(* Logix 5000 project; controller ACMI_PLC vendor 1 type 14 code 101 rev 19.11; software revision 19.01; part 8 of 9 *)
(* tags used below, declared in another part *)
   A : DINT;
   ACMI_BR_CNT : DINT;
   ACMI_Stat_Size : INT;
   ACMI_TO_CNT : DINT;
   ADCA : DINT;
   ADCB : DINT;
   B : DINT;
   Beam_MaxQ : DINT;
   Beam_MinQ : DINT;
   Beam_Q : DINT;
   BR_Stack : DINT[7200];
   BR_Stack_MAX : DINT;
   BR_Stack_Sum : DINT;
   BR_Stack_Top : DINT;
   BSSS_CLOSED : ALIAS FOR PointIONet:7:I.Pt00Data;
   BYPASS_KEY : ALIAS FOR PointIONet:5:I.Pt07Data;
   FAULT_BEAM_BL : BOOL;
   FAULT_BEAM_HI : BOOL;
   FAULT_BEAM_LO : BOOL;
   FAULT_BR_ACC : BOOL;
   FAULT_CODE : DINT;
   FAULT_QOW1 : BOOL;
   FAULT_ST1_AB_HI : BOOL;
   FAULT_ST1_AB_LO : BOOL;
   FAULT_ST1_BA_HI : BOOL;
   FAULT_ST1_BA_LO : BOOL;
   FAULT_ST1_BLA : BOOL;
   FAULT_ST1_BLB : BOOL;
   FAULT_ST1_QAT : BOOL;
   FAULT_ST2_AB_HI : BOOL;
   FAULT_ST2_AB_LO : BOOL;
   FAULT_ST2_BA_HI : BOOL;
   FAULT_ST2_BA_LO : BOOL;
   FAULT_ST2_BLA : BOOL;
   FAULT_ST2_BLB : BOOL;
   FAULT_ST2_QAT : BOOL;
   FAULT_TO_ACC : BOOL;
   FAULT_TWB : BOOL;
   FAULT_WDT : BOOL;
   Initialize : BOOL;
   LBSS_CLOSED : ALIAS FOR PointIONet:7:I.Pt01Data;
   ST1_MaxQ : DINT;
   ST1_MinQ : DINT;
   ST1_QAB : DINT;
   ST1_QBA : DINT;
   ST2_MaxQ : DINT;
   ST2_MinQ : DINT;
   ST2_QAB : DINT;
   ST2_QBA : DINT;
   ST_HI_FAULT : BOOL;
   ST_LO_FAULT : BOOL;
   ST_Size : BOOL;
   ST_Type : BOOL;
   Stack_Size : DINT;
   TO_Cntr : COUNTER;
   TO_DISABLED : ALIAS FOR PointIONet:7:I.Pt03Data;
   TO_Stack : DINT[120];
   TO_Stack_MAX : DINT;
   TO_Stack_Size : DINT;
   TO_Stack_Sum : DINT;
   TO_Stack_Top : DINT;
   TO_Status_Error : BOOL;
   Update_ST1_QAB : BOOL;
   Update_ST1_QBA : BOOL;
   Update_ST2_QAB : BOOL;
   Update_ST2_QBA : BOOL;
   Zero : DINT[7200];

        [22].Hist[2930] := 1, [22].Hist[2938] := 1, [22].Hist[2946] := 1, [22].Hist[2954] := 1, [22].Hist[2962] := 1, [22].Hist[2970] := 1, [22].Hist[2975] := 1, [22].Hist[2978] := 1, [22].Hist[2986] := 1, [22].Hist[2994] := 1, [22].Hist[3002] := 1, [22].Hist[3010] := 1, [22].Hist[3018] := 1, [22].Hist[3026] := 1, [22].Hist[3034] := 1, [22].Hist[3042] := 1, [22].Hist[3050] := 1, [22].Hist[3058] := 1, [22].Hist[3066] := 1, [22].Hist[3074] := 1, [22].Hist[3082] := 1, [22].Hist[3090] := 1, [22].Hist[3098] := 1, [22].Hist[3106] := 1, [22].Hist[3114] := 1, [22].Hist[3122] := 1, [22].Hist[3130] := 1, [22].Hist[3138] := 1, [22].Hist[3146] := 1, [22].Hist[3152] := 1, [22].Hist[3154] := 1, [22].Hist[3162] := 1, [22].Hist[3170] := 1, [22].Hist[3178] := 1, [22].Hist[3181] := 1, [22].Hist[3186] := 1, [22].Hist[3194] := 1, [22].Hist[3202] := 1, [22].Hist[3210] := 1, [22].Hist[3218] := 1, [22].Hist[3226] := 1, [22].Hist[3234] := 1, [22].Hist[3242] := 1, [22].Hist[3250] := 1, [22].Hist[3258] := 1, [22].Hist[3266] := 1, [22].Hist[3274] := 1, [22].Hist[3282] := 1, [22].Hist[3290] := 1, [22].Hist[3298] := 1, [22].Hist[3306] := 1, [22].Hist[3314] := 1, [22].Hist[3322] := 1, [22].Hist[3330] := 1, [22].Hist[3333] := 1, [22].Hist[3338] := 1, [22].Hist[3346] := 1, [22].Hist[3354] := 1, [22].Hist[3362] := 1, [22].Hist[3370] := 1,
        [22].Hist[3378] := 1, [22].Hist[3386] := 1, [22].Hist[3394] := 1, [22].Hist[3402] := 1, [22].Hist[3410] := 1, [22].Hist[3418] := 1, [22].Hist[3420] := 1, [22].Hist[3426] := 1, [22].Hist[3434] := 1, [22].Hist[3442] := 1, [22].Hist[3450] := 1, [22].Hist[3458] := 1, [22].Hist[3466] := 1, [22].Hist[3474] := 1, [22].Hist[3482] := 1, [22].Hist[3490] := 1, [22].Hist[3497] := 1, [22].Hist[3498] := 1, [22].Hist[3506] := 1, [22].Hist[3514] := 1, [22].Hist[3522] := 1, [22].Hist[3530] := 1, [22].Hist[3538] := 1, [22].Hist[3546] := 1, [22].Hist[3554] := 1, [22].Hist[3562] := 1, [22].Hist[3570] := 1, [22].Hist[3578] := 1, [22].Hist[3586] := 1, [22].Hist[3594] := 1, [22].Hist[3602] := 1, [22].Hist[3610] := 1, [22].Hist[3618] := 1, [22].Hist[3626] := 1, [22].Hist[3634] := 1, [22].Hist[3642] := 1, [22].Hist[3650] := 1, [22].Hist[3658] := 1, [22].Hist[3666] := 1, [22].Hist[3674] := 1, [22].Hist[3682] := 1, [22].Hist[3690] := 1, [22].Hist[3698] := 1, [22].Hist[3706] := 1, [22].Hist[3714] := 1, [22].Hist[3722] := 1, [22].Hist[3730] := 1, [22].Hist[3738] := 1, [22].Hist[3746] := 1, [22].Hist[3754] := 1, [22].Hist[3762] := 1, [22].Hist[3770] := 1, [22].Hist[3778] := 1, [22].Hist[3786] := 1, [22].Hist[3794] := 1, [22].Hist[3802] := 1, [22].Hist[3810] := 1, [22].Hist[3818] := 1, [22].Hist[3826] := 1, [22].Hist[3834] := 1,
        [22].Hist[3842] := 1, [22].Hist[3850] := 1, [22].Hist[3858] := 1, [22].Hist[3866] := 1, [22].Hist[3874] := 1, [22].Hist[3882] := 1, [22].Hist[3890] := 1, [22].Hist[3898] := 1, [22].Hist[3906] := 1, [22].Hist[3914] := 1, [22].Hist[3922] := 1, [22].Hist[3924] := 1, [22].Hist[3930] := 1, [22].Hist[3938] := 1, [22].Hist[3946] := 1, [22].Hist[3954] := 1, [22].Hist[3962] := 1, [22].Hist[3970] := 1, [22].Hist[3978] := 1, [22].Hist[3986] := 1, [22].Hist[3994] := 1, [22].Hist[4002] := 1, [22].Hist[4010] := 1, [22].Hist[4018] := 1, [22].Hist[4026] := 1, [22].Hist[4034] := 1, [22].Hist[4042] := 1, [22].Hist[4045] := 1, [22].Hist[4050] := 1, [22].Hist[4058] := 1, [22].Hist[4066] := 1, [22].Hist[4074] := 1, [22].Hist[4082] := 1, [22].Hist[4090] := 1, [22].Top := 3955, [22].Sum := 539, [23].Hist[68] := 1, [23].Hist[123] := 1, [23].Hist[181] := 1, [23].Hist[417] := 1, [23].Hist[431] := 1, [23].Hist[488] := 1, [23].Hist[540] := 1, [23].Hist[567] := 1, [23].Hist[661] := 1, [23].Hist[805] := 1, [23].Hist[1153] := 1, [23].Hist[1377] := 1, [23].Hist[1435] := 1, [23].Hist[1727] := 1, [23].Hist[1773] := 1, [23].Hist[1817] := 1, [23].Hist[2324] := 1, [23].Hist[2512] := 1, [23].Hist[2756] := 1, [23].Hist[2975] := 1, [23].Hist[3152] := 1, [23].Hist[3181] := 1, [23].Hist[3333] := 1, [23].Hist[3420] := 1,
        [23].Hist[3497] := 1, [23].Hist[3924] := 1, [23].Hist[4045] := 1, [23].Top := 3955, [23].Sum := 27);
   Bx : DINT; {access Read Only}
   Data_Type : BOOL := 1;
   DrdyTimer : TIMER := (PRE := 500, ACC := 200, EN := 1, TT := 1);
   DrdyWDT : DINT := 220;
   ev_num : COUNTER := (ACC := 866343322, DN := 1);
   Fit_Linear_1 : DINT := 91449; {constant}
   Fit_Linear_2 : DINT := 10000; {constant}
   Fit_Off : DINT := 7; {constant}
   Fit_Quad_1 : DINT := 219; {constant}
   Fit_Quad_2 : DINT := 1000000; {constant}
   Hist : BOOL[4096] := ([956] := 1, [1408] := 1, [2824] := 1, [3245] := 1, [3333] := 1, [3825] := 1, [4017] := 1);
   index : DINT;
   NewData : BOOL := 1;
   Q : DINT := 15921;
   QIW : BOOL := 1;
   Qlinear : DINT := 15299;
   QOW_FailSafe : TIMER := (PRE := 2000, ACC := 340); {access Read Only}
   QOW_Latch : BOOL;
   Qquad : DINT := 615;
   ReadData : BOOL;
   Relay_Status : ALIAS FOR PointIONet:5:I.Pt04Data;
   Safety_Shutters : BOOL;
   ST1AB_ADCA : DINT := 64; {access Read Only}
   ST1AB_ADCB : DINT := 3; {access Read Only}
   ST1BA_ADCA : DINT := -1; {access Read Only}
   ST1BA_ADCB : DINT := 62; {access Read Only}
   ST2AB_ADCA : DINT := 1692; {access Read Only}
   ST2AB_ADCB : DINT := 3; {access Read Only}
   ST2BA_ADCA : DINT; {access Read Only}
   ST2BA_ADCB : DINT := 1673; {access Read Only}
   Stack_Data : DINT := 180;
   STQ : DINT := 15921; {access Read Only}
   STQmax : DINT := 16400; {access Read Only}
   STQmin : DINT := 15400; {access Read Only}
   Sum : INT := 7;
   Toggle : BitStat[12];
   Top : INT := 361;
   TWB_FailSafe : TIMER := (PRE := 2000, ACC := 20); {access Read Only}
   TWB_Latch : BOOL;
   Update_Latch : BOOL := 1; {access Read Only}
   Update_Unlatch : BOOL; {access Read Only}
   w1 : DINT; {access Read Only}
   w2 : DINT; {access Read Only}
   WDT_Event_Limit : DINT := 265; {constant, access Read Only}
   x : DINT := 1673;
   y : DINT;
   z : DINT := 1673;
   z2 : DINT;
END_VAR

ROUTINE Bit_Toggle   (* ladder *)
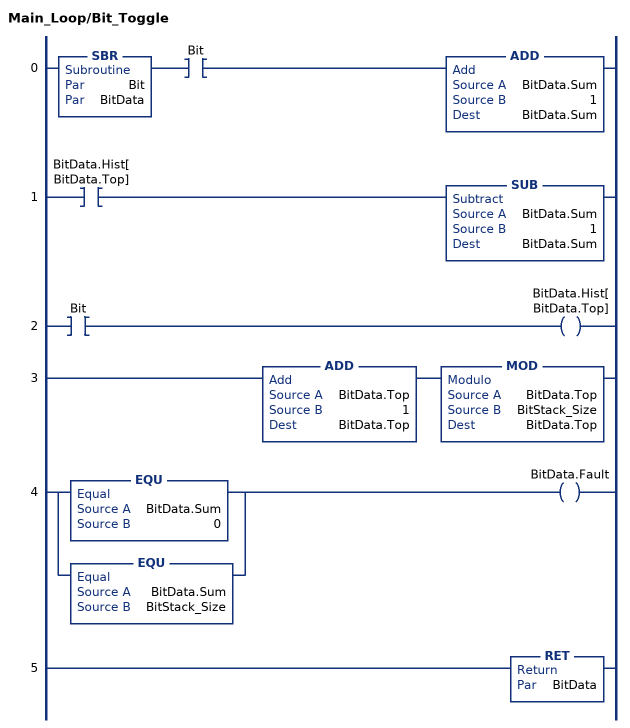
   [picture p14: Main_Loop/Bit_Toggle rungs 0-5]
   0: SBR(Bit,BitData)XIC(Bit)ADD(BitData.Sum,1,BitData.Sum);
   1: XIC(BitData.Hist[BitData.Top])SUB(BitData.Sum,1,BitData.Sum);
   2: XIC(Bit)OTE(BitData.Hist[BitData.Top]);
   3: ADD(BitData.Top,1,BitData.Top)MOD(BitData.Top,BitStack_Size,BitData.Top);
   4: [EQU(BitData.Sum,0) ,EQU(BitData.Sum,BitStack_Size) ]OTE(BitData.Fault);
   5: RET(BitData);
END_ROUTINE

ROUTINE Calc_Q   (* ladder *)
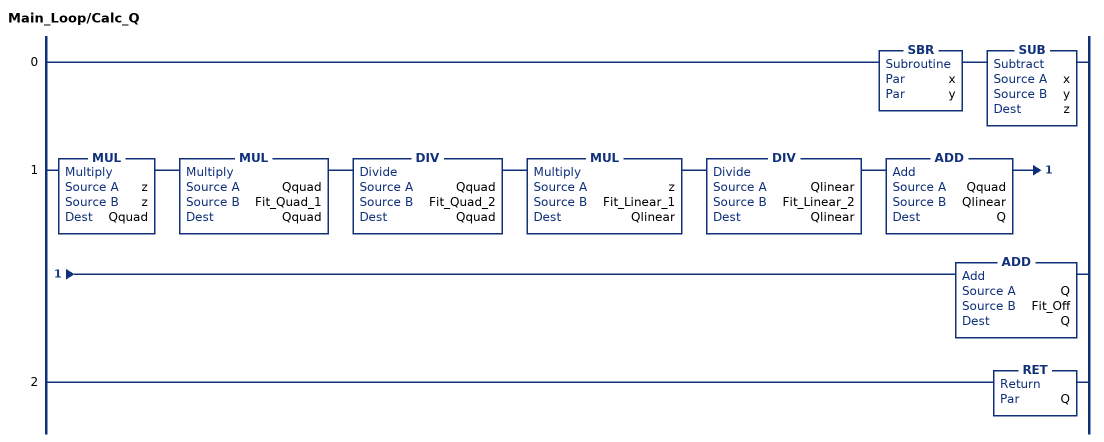
   0: SBR(x,y)SUB(x,y,z);
   1: MUL(z,z,Qquad)MUL(Qquad,Fit_Quad_1,Qquad)DIV(Qquad,Fit_Quad_2,Qquad)MUL(z,Fit_Linear_1,Qlinear)DIV(Qlinear,Fit_Linear_2,Qlinear)ADD(Qquad,Qlinear,Q)ADD(Q,Fit_Off,Q);
   2: RET(Q);
END_ROUTINE

ROUTINE MainRoutine   (* ladder *)
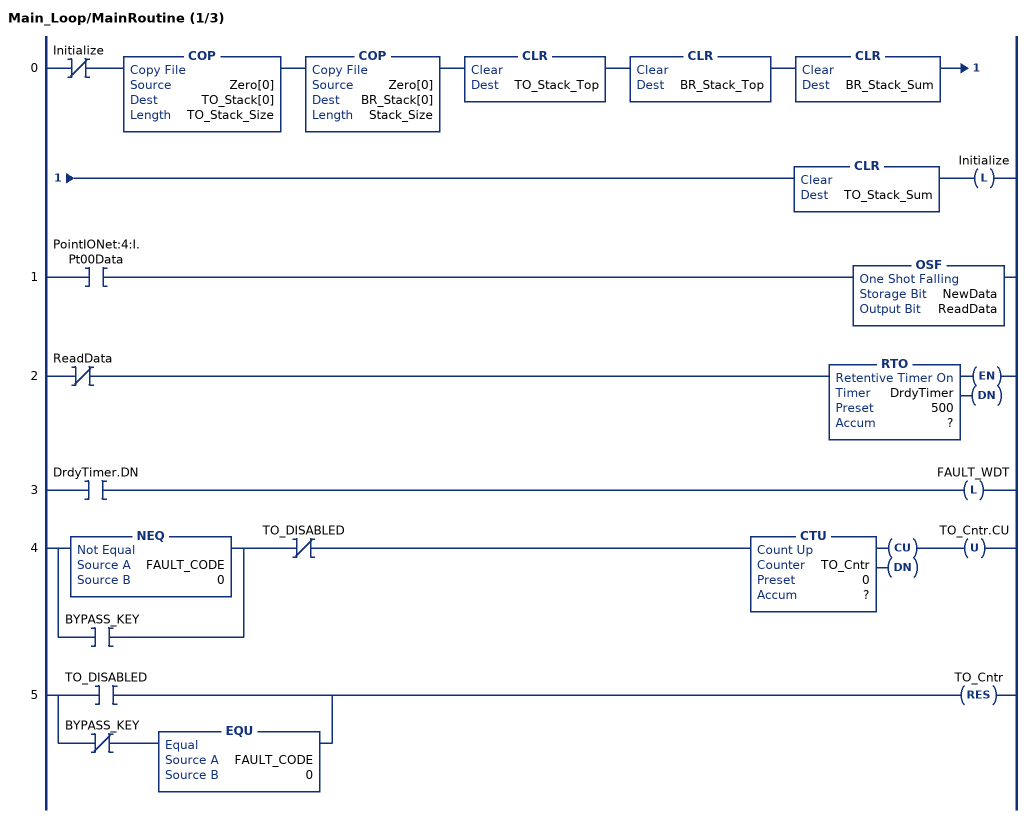
   0: XIO(Initialize)COP(Zero[0],TO_Stack[0],TO_Stack_Size)COP(Zero[0],BR_Stack[0],Stack_Size)CLR(TO_Stack_Top)CLR(BR_Stack_Top)CLR(BR_Stack_Sum)CLR(TO_Stack_Sum)OTL(Initialize);
   1: XIC(PointIONet:4:I.Pt00Data)OSF(NewData,ReadData);
   2: XIO(ReadData)RTO(DrdyTimer,?,?);
   3: XIC(DrdyTimer.DN)OTL(FAULT_WDT);
   4: [NEQ(FAULT_CODE,0) ,XIC(BYPASS_KEY) ]XIO(TO_DISABLED)CTU(TO_Cntr,?,?)OTU(TO_Cntr.CU);
   5: [XIC(TO_DISABLED) ,XIO(BYPASS_KEY) EQU(FAULT_CODE,0) ]RES(TO_Cntr);
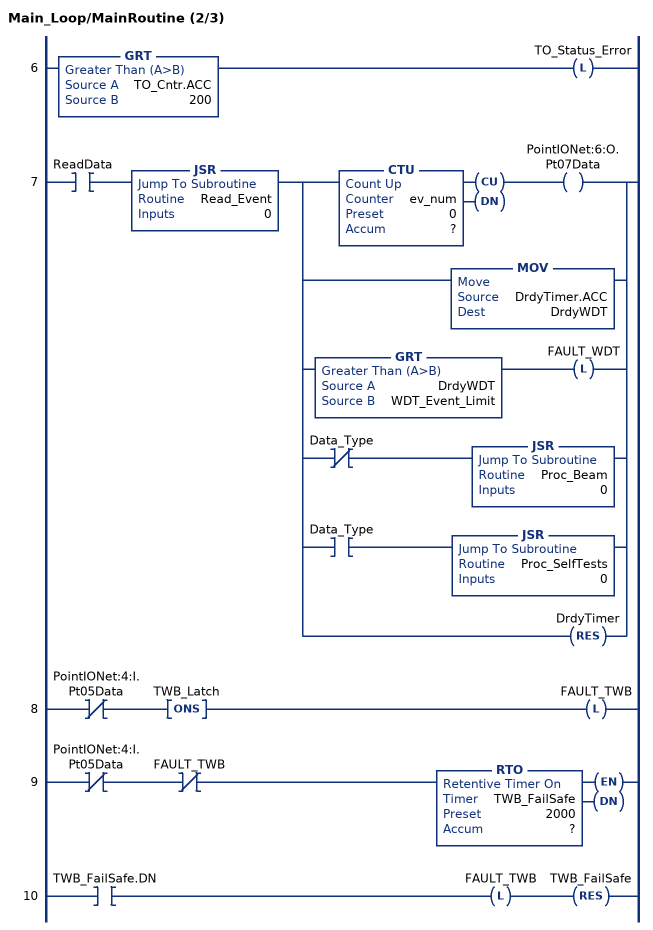
   6: GRT(TO_Cntr.ACC,200)OTL(TO_Status_Error);
   7: XIC(ReadData)JSR(Read_Event,0)[CTU(ev_num,?,?) OTE(PointIONet:6:O.Pt07Data) ,MOV(DrdyTimer.ACC,DrdyWDT) ,GRT(DrdyWDT,WDT_Event_Limit) OTL(FAULT_WDT) ,XIO(Data_Type) JSR(Proc_Beam,0) ,XIC(Data_Type) JSR(Proc_SelfTests,0) ,RES(DrdyTimer) ];
   8: XIO(PointIONet:4:I.Pt05Data)ONS(TWB_Latch)OTL(FAULT_TWB);
   9: XIO(PointIONet:4:I.Pt05Data)XIO(FAULT_TWB)RTO(TWB_FailSafe,?,?);
   10: XIC(TWB_FailSafe.DN)OTL(FAULT_TWB)RES(TWB_FailSafe);
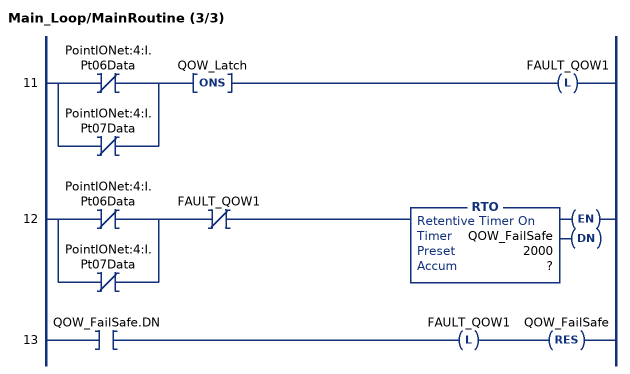
   11: [XIO(PointIONet:4:I.Pt06Data) ,XIO(PointIONet:4:I.Pt07Data) ]ONS(QOW_Latch)OTL(FAULT_QOW1);
   12: [XIO(PointIONet:4:I.Pt06Data) ,XIO(PointIONet:4:I.Pt07Data) ]XIO(FAULT_QOW1)RTO(QOW_FailSafe,?,?);
   13: XIC(QOW_FailSafe.DN)OTL(FAULT_QOW1)RES(QOW_FailSafe);
END_ROUTINE

ROUTINE Proc_Beam   (* ladder *)
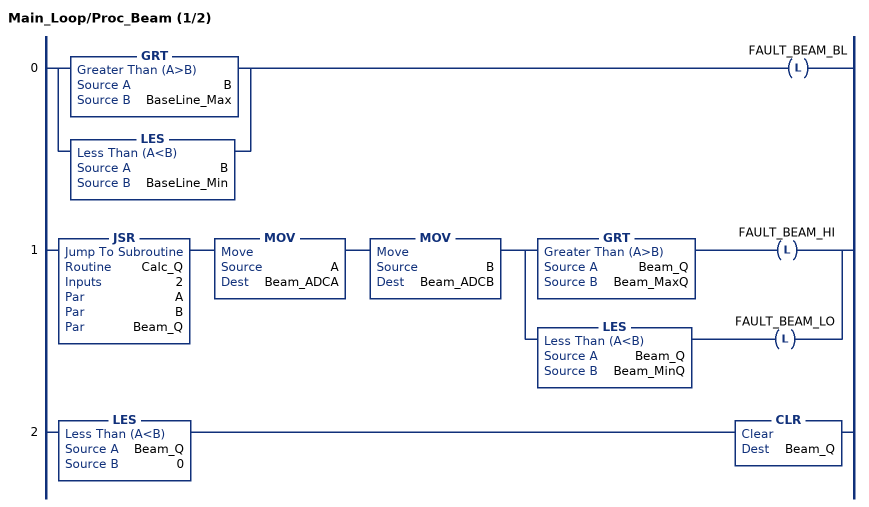
   0: [GRT(B,BaseLine_Max) ,LES(B,BaseLine_Min) ]OTL(FAULT_BEAM_BL);
   1: JSR(Calc_Q,2,A,B,Beam_Q)MOV(A,Beam_ADCA)MOV(B,Beam_ADCB)[GRT(Beam_Q,Beam_MaxQ) OTL(FAULT_BEAM_HI) ,LES(Beam_Q,Beam_MinQ) OTL(FAULT_BEAM_LO) ];
   2: LES(Beam_Q,0)CLR(Beam_Q);
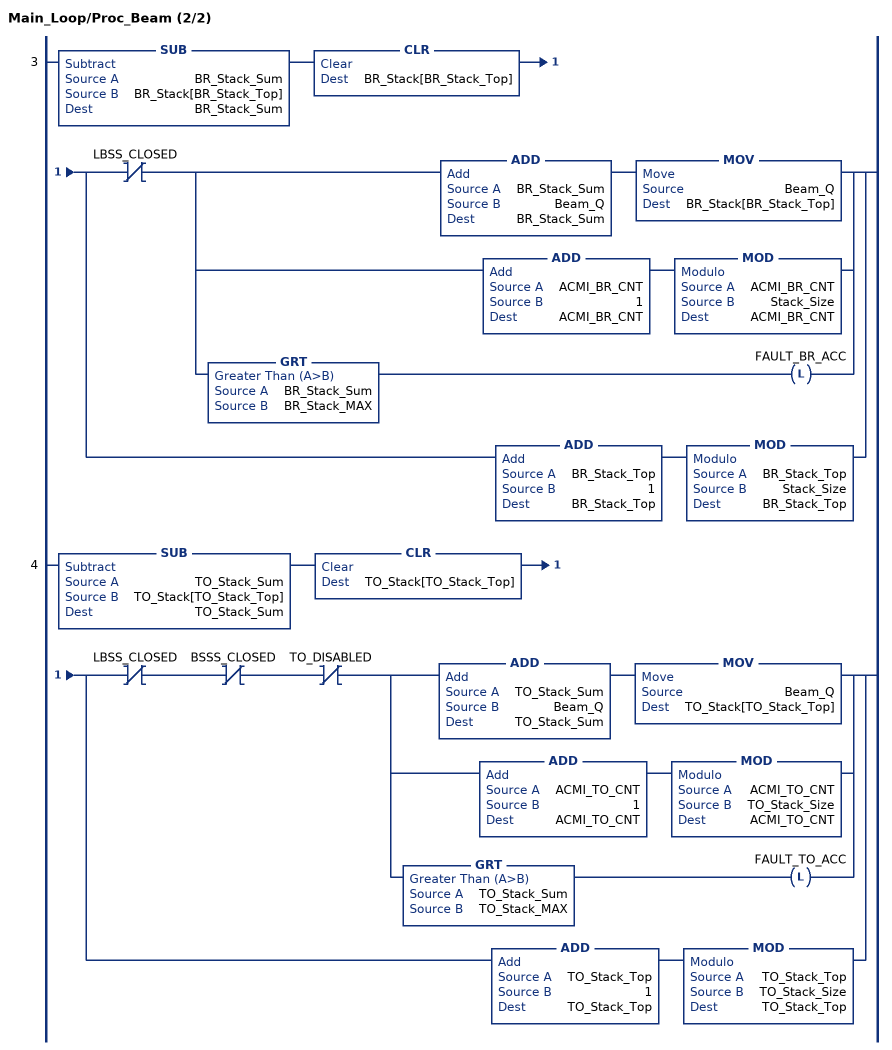
   3: SUB(BR_Stack_Sum,BR_Stack[BR_Stack_Top],BR_Stack_Sum)CLR(BR_Stack[BR_Stack_Top])[XIO(LBSS_CLOSED) [ADD(BR_Stack_Sum,Beam_Q,BR_Stack_Sum) MOV(Beam_Q,BR_Stack[BR_Stack_Top]) ,ADD(ACMI_BR_CNT,1,ACMI_BR_CNT) MOD(ACMI_BR_CNT,Stack_Size,ACMI_BR_CNT) ,GRT(BR_Stack_Sum,BR_Stack_MAX) OTL(FAULT_BR_ACC) ] ,ADD(BR_Stack_Top,1,BR_Stack_Top) MOD(BR_Stack_Top,Stack_Size,BR_Stack_Top) ];
   4: SUB(TO_Stack_Sum,TO_Stack[TO_Stack_Top],TO_Stack_Sum)CLR(TO_Stack[TO_Stack_Top])[XIO(LBSS_CLOSED) XIO(BSSS_CLOSED) XIO(TO_DISABLED) [ADD(TO_Stack_Sum,Beam_Q,TO_Stack_Sum) MOV(Beam_Q,TO_Stack[TO_Stack_Top]) ,ADD(ACMI_TO_CNT,1,ACMI_TO_CNT) MOD(ACMI_TO_CNT,TO_Stack_Size,ACMI_TO_CNT) ,GRT(TO_Stack_Sum,TO_Stack_MAX) OTL(FAULT_TO_ACC) ] ,ADD(TO_Stack_Top,1,TO_Stack_Top) MOD(TO_Stack_Top,TO_Stack_Size,TO_Stack_Top) ];
END_ROUTINE

ROUTINE Proc_SelfTests   (* ladder *)
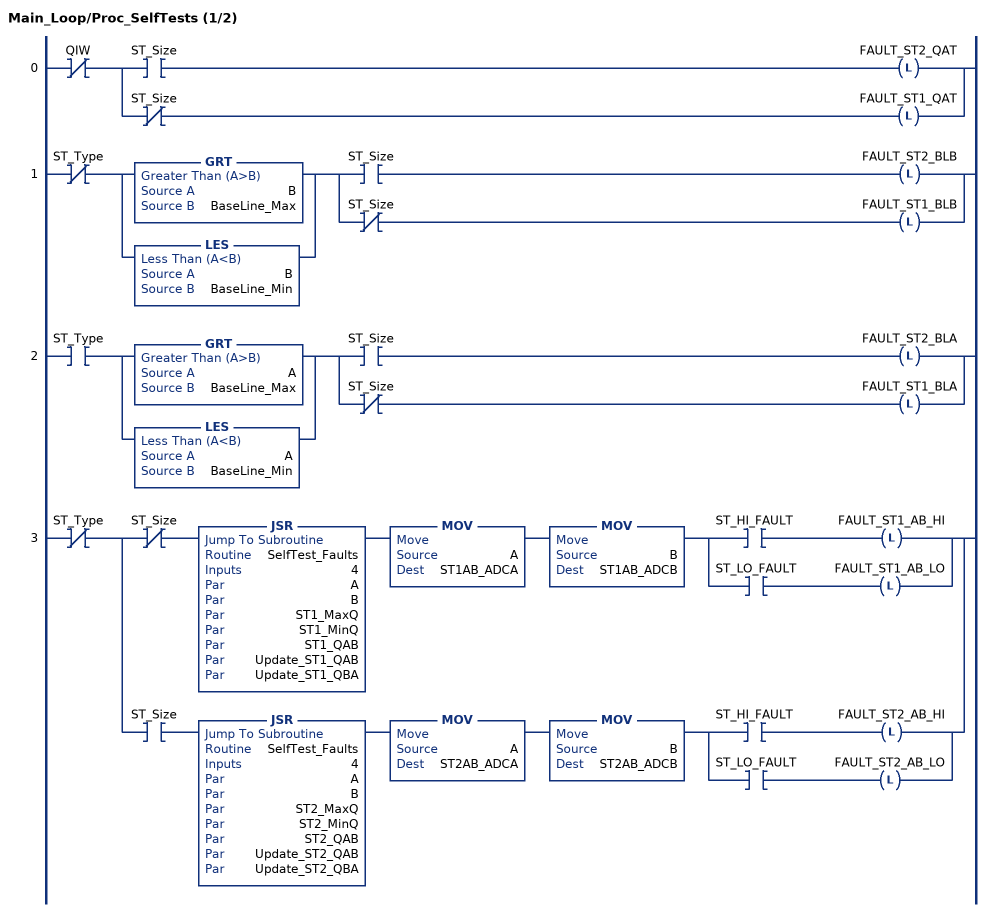
   0: XIO(QIW)[XIC(ST_Size) OTL(FAULT_ST2_QAT) ,XIO(ST_Size) OTL(FAULT_ST1_QAT) ];
   1: XIO(ST_Type)[GRT(B,BaseLine_Max) ,LES(B,BaseLine_Min) ][XIC(ST_Size) OTL(FAULT_ST2_BLB) ,XIO(ST_Size) OTL(FAULT_ST1_BLB) ];
   2: XIC(ST_Type)[GRT(A,BaseLine_Max) ,LES(A,BaseLine_Min) ][XIC(ST_Size) OTL(FAULT_ST2_BLA) ,XIO(ST_Size) OTL(FAULT_ST1_BLA) ];
   3: XIO(ST_Type)[XIO(ST_Size) JSR(SelfTest_Faults,4,A,B,ST1_MaxQ,ST1_MinQ,ST1_QAB,Update_ST1_QAB,Update_ST1_QBA) MOV(A,ST1AB_ADCA) MOV(B,ST1AB_ADCB) [XIC(ST_HI_FAULT) OTL(FAULT_ST1_AB_HI) ,XIC(ST_LO_FAULT) OTL(FAULT_ST1_AB_LO) ] ,XIC(ST_Size) JSR(SelfTest_Faults,4,A,B,ST2_MaxQ,ST2_MinQ,ST2_QAB,Update_ST2_QAB,Update_ST2_QBA) MOV(A,ST2AB_ADCA) MOV(B,ST2AB_ADCB) [XIC(ST_HI_FAULT) OTL(FAULT_ST2_AB_HI) ,XIC(ST_LO_FAULT) OTL(FAULT_ST2_AB_LO) ] ];
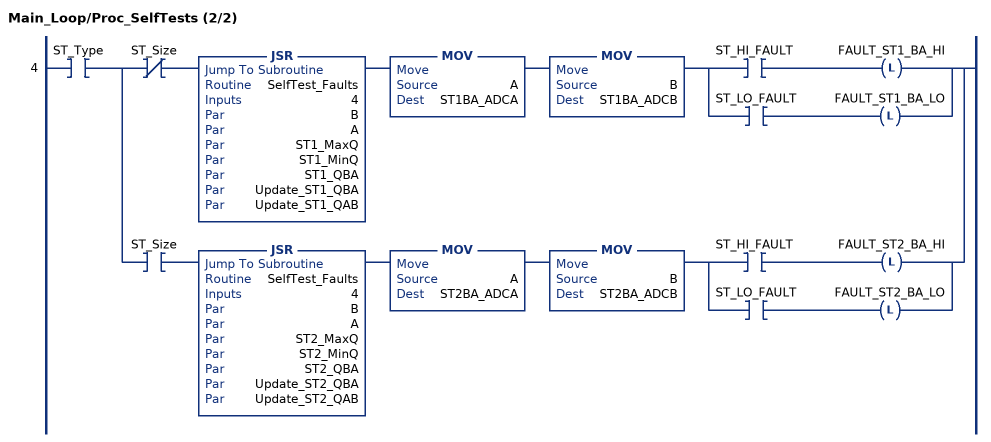
   4: XIC(ST_Type)[XIO(ST_Size) JSR(SelfTest_Faults,4,B,A,ST1_MaxQ,ST1_MinQ,ST1_QBA,Update_ST1_QBA,Update_ST1_QAB) MOV(A,ST1BA_ADCA) MOV(B,ST1BA_ADCB) [XIC(ST_HI_FAULT) OTL(FAULT_ST1_BA_HI) ,XIC(ST_LO_FAULT) OTL(FAULT_ST1_BA_LO) ] ,XIC(ST_Size) JSR(SelfTest_Faults,4,B,A,ST2_MaxQ,ST2_MinQ,ST2_QBA,Update_ST2_QBA,Update_ST2_QAB) MOV(A,ST2BA_ADCA) MOV(B,ST2BA_ADCB) [XIC(ST_HI_FAULT) OTL(FAULT_ST2_BA_HI) ,XIC(ST_LO_FAULT) OTL(FAULT_ST2_BA_LO) ] ];
END_ROUTINE

ROUTINE Read_Event   (* ladder *)
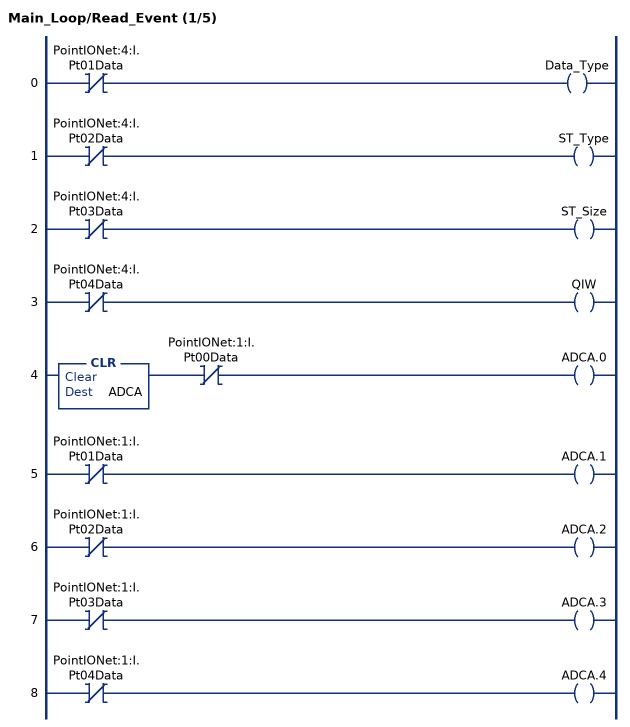
   0: XIO(PointIONet:4:I.Pt01Data)OTE(Data_Type);
   1: XIO(PointIONet:4:I.Pt02Data)OTE(ST_Type);
   2: XIO(PointIONet:4:I.Pt03Data)OTE(ST_Size);
   3: XIO(PointIONet:4:I.Pt04Data)OTE(QIW);
   4: CLR(ADCA)XIO(PointIONet:1:I.Pt00Data)OTE(ADCA.0);
   5: XIO(PointIONet:1:I.Pt01Data)OTE(ADCA.1);
   6: XIO(PointIONet:1:I.Pt02Data)OTE(ADCA.2);
   7: XIO(PointIONet:1:I.Pt03Data)OTE(ADCA.3);
   8: XIO(PointIONet:1:I.Pt04Data)OTE(ADCA.4);
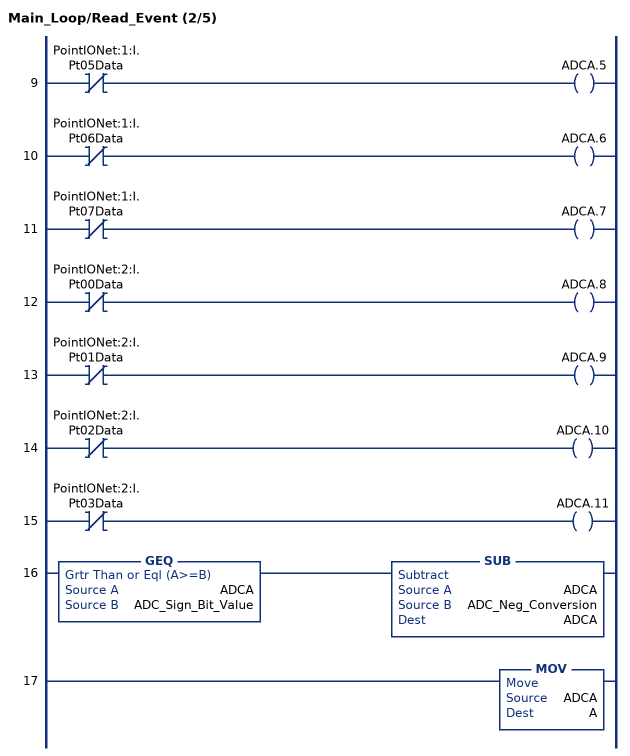
   9: XIO(PointIONet:1:I.Pt05Data)OTE(ADCA.5);
   10: XIO(PointIONet:1:I.Pt06Data)OTE(ADCA.6);
   11: XIO(PointIONet:1:I.Pt07Data)OTE(ADCA.7);
   12: XIO(PointIONet:2:I.Pt00Data)OTE(ADCA.8);
   13: XIO(PointIONet:2:I.Pt01Data)OTE(ADCA.9);
   14: XIO(PointIONet:2:I.Pt02Data)OTE(ADCA.10);
   15: XIO(PointIONet:2:I.Pt03Data)OTE(ADCA.11);
   16: GEQ(ADCA,ADC_Sign_Bit_Value)SUB(ADCA,ADC_Neg_Conversion,ADCA);
   17: MOV(ADCA,A);
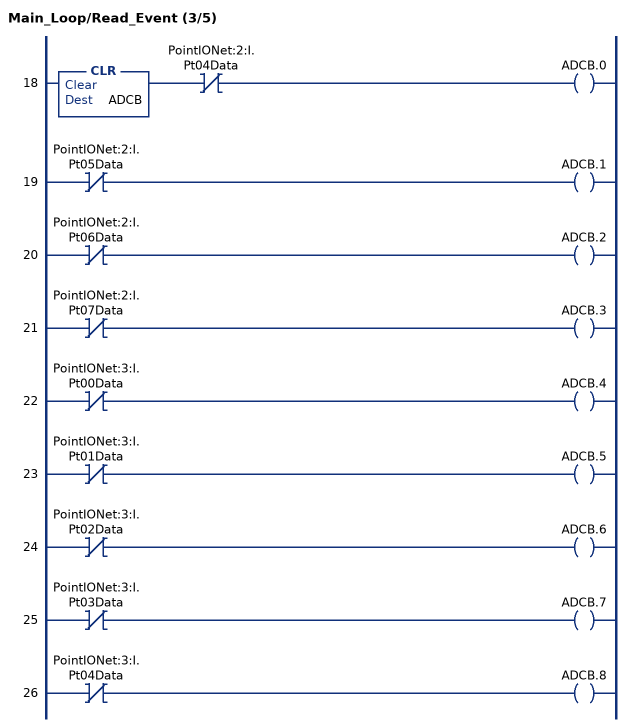
   18: CLR(ADCB)XIO(PointIONet:2:I.Pt04Data)OTE(ADCB.0);
   19: XIO(PointIONet:2:I.Pt05Data)OTE(ADCB.1);
   20: XIO(PointIONet:2:I.Pt06Data)OTE(ADCB.2);
   21: XIO(PointIONet:2:I.Pt07Data)OTE(ADCB.3);
   22: XIO(PointIONet:3:I.Pt00Data)OTE(ADCB.4);
   23: XIO(PointIONet:3:I.Pt01Data)OTE(ADCB.5);
   24: XIO(PointIONet:3:I.Pt02Data)OTE(ADCB.6);
   25: XIO(PointIONet:3:I.Pt03Data)OTE(ADCB.7);
   26: XIO(PointIONet:3:I.Pt04Data)OTE(ADCB.8);
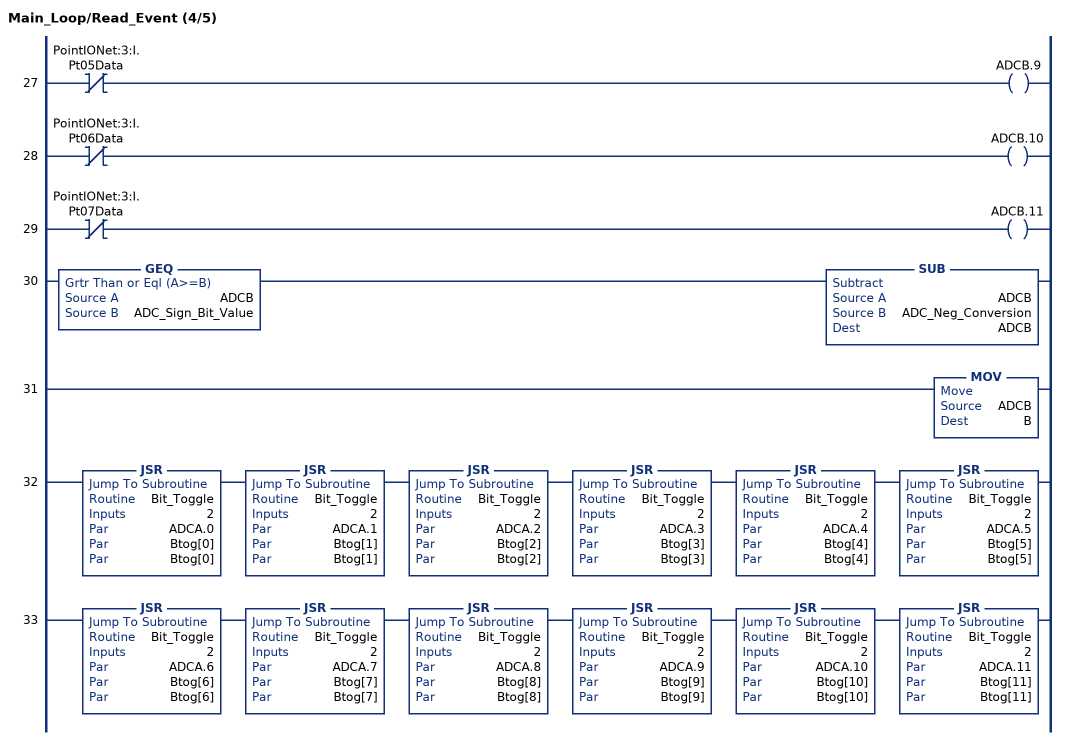
   27: XIO(PointIONet:3:I.Pt05Data)OTE(ADCB.9);
   28: XIO(PointIONet:3:I.Pt06Data)OTE(ADCB.10);
   29: XIO(PointIONet:3:I.Pt07Data)OTE(ADCB.11);
   30: GEQ(ADCB,ADC_Sign_Bit_Value)SUB(ADCB,ADC_Neg_Conversion,ADCB);
   31: MOV(ADCB,B);
   32: JSR(Bit_Toggle,2,ADCA.0,Btog[0],Btog[0])JSR(Bit_Toggle,2,ADCA.1,Btog[1],Btog[1])JSR(Bit_Toggle,2,ADCA.2,Btog[2],Btog[2])JSR(Bit_Toggle,2,ADCA.3,Btog[3],Btog[3])JSR(Bit_Toggle,2,ADCA.4,Btog[4],Btog[4])JSR(Bit_Toggle,2,ADCA.5,Btog[5],Btog[5]);
   33: JSR(Bit_Toggle,2,ADCA.6,Btog[6],Btog[6])JSR(Bit_Toggle,2,ADCA.7,Btog[7],Btog[7])JSR(Bit_Toggle,2,ADCA.8,Btog[8],Btog[8])JSR(Bit_Toggle,2,ADCA.9,Btog[9],Btog[9])JSR(Bit_Toggle,2,ADCA.10,Btog[10],Btog[10])JSR(Bit_Toggle,2,ADCA.11,Btog[11],Btog[11]);
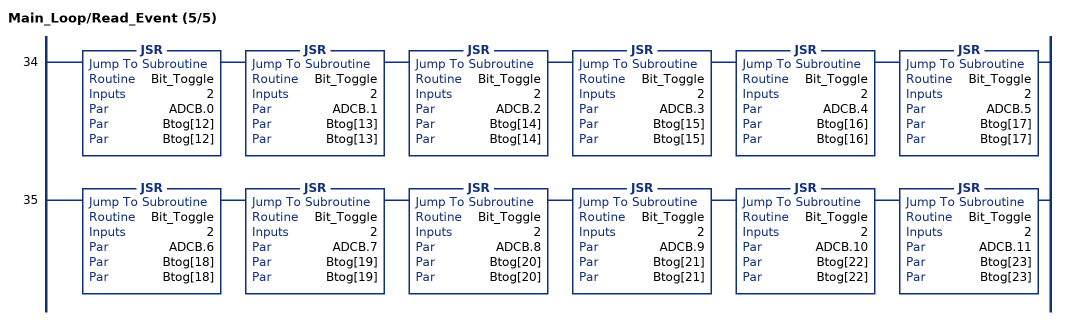
   34: JSR(Bit_Toggle,2,ADCB.0,Btog[12],Btog[12])JSR(Bit_Toggle,2,ADCB.1,Btog[13],Btog[13])JSR(Bit_Toggle,2,ADCB.2,Btog[14],Btog[14])JSR(Bit_Toggle,2,ADCB.3,Btog[15],Btog[15])JSR(Bit_Toggle,2,ADCB.4,Btog[16],Btog[16])JSR(Bit_Toggle,2,ADCB.5,Btog[17],Btog[17]);
   35: JSR(Bit_Toggle,2,ADCB.6,Btog[18],Btog[18])JSR(Bit_Toggle,2,ADCB.7,Btog[19],Btog[19])JSR(Bit_Toggle,2,ADCB.8,Btog[20],Btog[20])JSR(Bit_Toggle,2,ADCB.9,Btog[21],Btog[21])JSR(Bit_Toggle,2,ADCB.10,Btog[22],Btog[22])JSR(Bit_Toggle,2,ADCB.11,Btog[23],Btog[23]);
END_ROUTINE

ROUTINE SelfTest_Faults   (* ladder *)
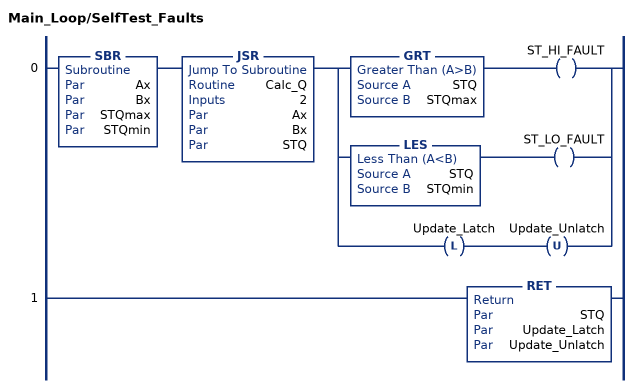
   0: SBR(Ax,Bx,STQmax,STQmin)JSR(Calc_Q,2,Ax,Bx,STQ)[GRT(STQ,STQmax) OTE(ST_HI_FAULT) ,LES(STQ,STQmin) OTE(ST_LO_FAULT) ,OTL(Update_Latch) OTU(Update_Unlatch) ];
   1: RET(STQ,Update_Latch,Update_Unlatch);
END_ROUTINE
END_PROGRAM

PROGRAM MainProgram   (* main routine Self_Test_Stats *)
VAR
   A_AVG : REAL := 2047.0;
   A_HIST : DINT[50] := ([0] := 2047, [1] := 2047, [2] := 2047, [3] := 2047, [4] := 2047, [5] := 2047, [6] := 2047, [7] := 2047, [8] := 2047, [9] := 2047, [10] := 2047, [11] := 2047, [12] := 2047, [13] := 2047, [14] := 2047, [15] := 2047, [16] := 2047, [17] := 2047, [18] := 2047, [19] := 2047, [20] := 2047, [21] := 2047, [22] := 2047, [23] := 2047, [24] := 2047, [25] := 2047, [26] := 2047, [27] := 2047, [28] := 2047, [29] := 2047, [30] := 2047, [31] := 2047, [32] := 2047, [33] := 2047, [34] := 2047, [35] := 2047, [36] := 2047, [37] := 2047, [38] := 2047, [39] := 2047, [40] := 2047, [41] := 2047, [42] := 2047, [43] := 2047, [44] := 2047, [45] := 2047, [46] := 2047, [47] := 2047, [48] := 2047, [49] := 2047);
   A_SUM : DINT := 102350;
   A_TOP : SINT := 33;
   AB_N : SINT := 50;
   ACMI_ST1_QAB_VAR : REAL := 25.50509;
   ACMI_ST1_QBA_VAR : REAL := 25.955812;
   ACMI_ST2_QAB_VAR : REAL := 25.458477;
   ACMI_ST2_QBA_VAR : REAL := 26.01466;
   ADC1 : COUNTER;
   B_AVG : REAL := 55.1;
   B_HIST : DINT[50] := ([0] := 56, [1] := 62, [2] := 59, [3] := 45, [4] := 58, [5] := 53, [6] := 53, [7] := 69, [8] := 56, [9] := 57, [10] := 47, [11] := 56, [12] := 53, [13] := 39, [14] := 43, [15] := 31, [16] := 69, [17] := 48, [18] := 47, [19] := 55, [20] := 44, [21] := 40, [22] := 38, [23] := 60, [24] := 73, [25] := 68, [26] := 48, [27] := 49, [28] := 53, [29] := 44, [30] := 69, [31] := 71, [32] := 64, [33] := 66, [34] := 69, [35] := 54, [36] := 53, [37] := 47, [38] := 50, [39] := 53, [40] := 53, [41] := 73, [42] := 59, [43] := 64, [44] := 62, [45] := 48, [46] := 56, [47] := 38, [48] := 76, [49] := 57);
   B_SUM : DINT := 2755;
   B_TOP : SINT := 33;
   Bin_Width : REAL := 0.015; {constant}
   C_AVG : REAL := 41.1; {access Read Only}
   C_HIST : DINT[50] := ([0] := 45, [1] := 43, [2] := 40, [3] := 32, [4] := 46, [5] := 31, [6] := 55, [7] := 37, [8] := 48, [9] := 49, [10] := 31, [11] := 27, [12] := 36, [13] := 33, [14] := 48, [15] := 43, [16] := 34, [17] := 39, [18] := 32, [19] := 41, [20] := 33, [21] := 35, [22] := 55, [23] := 43, [24] := 45, [25] := 34, [26] := 46, [27] := 30, [28] := 30, [29] := 58, [30] := 46, [31] := 51, [32] := 49, [33] := 50, [34] := 53, [35] := 35, [36] := 48, [37] := 40, [38] := 38, [39] := 30, [40] := 46, [41] := 47, [42] := 34, [43] := 41, [44] := 42, [45] := 42, [46] := 33, [47] := 60, [48] := 56, [49] := 38); {access Read Only}
   C_SUM : DINT := 2078; {access Read Only}
   C_TOP : SINT := 31; {access Read Only}
   CAL_INIT : BOOL;
   CAL_Zero : DINT[50]; {constant, access Read Only}
   CD_N : SINT := 50; {access Read Only}
   CLR_AB : BOOL := 1;
   CLR_CD : BOOL := 1;
   D_AVG : REAL := 2047.0; {access Read Only}
   D_HIST : DINT[50] := ([0] := 2047, [1] := 2047, [2] := 2047, [3] := 2047, [4] := 2047, [5] := 2047, [6] := 2047, [7] := 2047, [8] := 2047, [9] := 2047, [10] := 2047, [11] := 2047, [12] := 2047, [13] := 2047, [14] := 2047, [15] := 2047, [16] := 2047, [17] := 2047, [18] := 2047, [19] := 2047, [20] := 2047, [21] := 2047, [22] := 2047, [23] := 2047, [24] := 2047, [25] := 2047, [26] := 2047, [27] := 2047, [28] := 2047, [29] := 2047, [30] := 2047, [31] := 2047, [32] := 2047, [33] := 2047, [34] := 2047, [35] := 2047, [36] := 2047, [37] := 2047, [38] := 2047, [39] := 2047, [40] := 2047, [41] := 2047, [42] := 2047, [43] := 2047, [44] := 2047, [45] := 2047, [46] := 2047, [47] := 2047, [48] := 2047, [49] := 2047); {access Read Only}
   D_SUM : DINT := 102350; {access Read Only}
   D_TOP : SINT := 31; {access Read Only}
   EmptyHist : DINT[31]; {constant}
   H : DINT[31] := ([30] := 200);
   HCntr : REAL := 15.98;
   Index : INT := 30;
   INDX : INT[500] := ([0] := 30, [1] := 30, [2] := 30, [3] := 30, [4] := 30, [5] := 30, [6] := 30, [7] := 30, [8] := 30, [9] := 30, [10] := 30, [11] := 30, [12] := 30, [13] := 30, [14] := 30, [15] := 30, [16] := 30, [17] := 30, [18] := 30, [19] := 30, [20] := 30, [21] := 30, [22] := 30, [23] := 30, [24] := 30, [25] := 30, [26] := 30, [27] := 30, [28] := 30, [29] := 30, [30] := 30, [31] := 30, [32] := 30, [33] := 30, [34] := 30, [35] := 30, [36] := 30, [37] := 30, [38] := 30, [39] := 30, [40] := 30, [41] := 30, [42] := 30, [43] := 30, [44] := 30, [45] := 30, [46] := 30, [47] := 30, [48] := 30, [49] := 30, [50] := 30, [51] := 30, [52] := 30, [53] := 30, [54] := 30, [55] := 30, [56] := 30, [57] := 30, [58] := 30, [59] := 30,
        [60] := 30, [61] := 30, [62] := 30, [63] := 30, [64] := 30, [65] := 30, [66] := 30, [67] := 30, [68] := 30, [69] := 30, [70] := 30, [71] := 30, [72] := 30, [73] := 30, [74] := 30, [75] := 30, [76] := 30, [77] := 30, [78] := 30, [79] := 30, [80] := 30, [81] := 30, [82] := 30, [83] := 30, [84] := 30, [85] := 30, [86] := 30, [87] := 30, [88] := 30, [89] := 30, [90] := 30, [91] := 30, [92] := 30, [93] := 30, [94] := 30, [95] := 30, [96] := 30, [97] := 30, [98] := 30, [99] := 30, [100] := 30, [101] := 30, [102] := 30, [103] := 30, [104] := 30, [105] := 30, [106] := 30, [107] := 30, [108] := 30, [109] := 30, [110] := 30, [111] := 30, [112] := 30, [113] := 30, [114] := 30, [115] := 30, [116] := 30, [117] := 30, [118] := 30, [119] := 30,
        [120] := 30, [121] := 30, [122] := 30, [123] := 30, [124] := 30, [125] := 30, [126] := 30, [127] := 30, [128] := 30, [129] := 30, [130] := 30, [131] := 30, [132] := 30, [133] := 30, [134] := 30, [135] := 30, [136] := 30, [137] := 30, [138] := 30, [139] := 30, [140] := 30, [141] := 30, [142] := 30, [143] := 30, [144] := 30, [145] := 30, [146] := 30, [147] := 30, [148] := 30, [149] := 30, [150] := 30, [151] := 30, [152] := 30, [153] := 30, [154] := 30, [155] := 30, [156] := 30, [157] := 30, [158] := 30, [159] := 30, [160] := 30, [161] := 30, [162] := 30, [163] := 30, [164] := 30, [165] := 30, [166] := 30, [167] := 30, [168] := 30, [169] := 30, [170] := 30, [171] := 30, [172] := 30, [173] := 30, [174] := 30, [175] := 30, [176] := 30, [177] := 30, [178] := 30, [179] := 30,
        [180] := 30, [181] := 30, [182] := 30, [183] := 30, [184] := 30, [185] := 30, [186] := 30, [187] := 30, [188] := 30, [189] := 30, [190] := 30, [191] := 30, [192] := 30, [193] := 30, [194] := 30, [195] := 30, [196] := 30, [197] := 30, [198] := 30, [199] := 30, [200] := -1, [201] := -1, [202] := -1, [203] := -1, [204] := -1, [205] := -1, [206] := -1, [207] := -1, [208] := -1, [209] := -1, [210] := -1, [211] := -1, [212] := -1, [213] := -1, [214] := -1, [215] := -1, [216] := -1, [217] := -1, [218] := -1, [219] := -1, [220] := -1, [221] := -1, [222] := -1, [223] := -1, [224] := -1, [225] := -1, [226] := -1, [227] := -1, [228] := -1, [229] := -1, [230] := -1, [231] := -1, [232] := -1, [233] := -1, [234] := -1, [235] := -1, [236] := -1, [237] := -1, [238] := -1, [239] := -1,
        [240] := -1, [241] := -1, [242] := -1, [243] := -1, [244] := -1, [245] := -1, [246] := -1, [247] := -1, [248] := -1, [249] := -1, [250] := -1, [251] := -1, [252] := -1, [253] := -1, [254] := -1, [255] := -1, [256] := -1, [257] := -1, [258] := -1, [259] := -1, [260] := -1, [261] := -1, [262] := -1, [263] := -1, [264] := -1, [265] := -1, [266] := -1, [267] := -1, [268] := -1, [269] := -1, [270] := -1, [271] := -1, [272] := -1, [273] := -1, [274] := -1, [275] := -1, [276] := -1, [277] := -1, [278] := -1, [279] := -1, [280] := -1, [281] := -1, [282] := -1, [283] := -1, [284] := -1, [285] := -1, [286] := -1, [287] := -1, [288] := -1, [289] := -1, [290] := -1, [291] := -1, [292] := -1, [293] := -1, [294] := -1, [295] := -1, [296] := -1, [297] := -1, [298] := -1, [299] := -1,
        [300] := -1, [301] := -1);
   Init_INDX : INT[500] := ([0] := -1, [1] := -1, [2] := -1, [3] := -1, [4] := -1, [5] := -1, [6] := -1, [7] := -1, [8] := -1, [9] := -1, [10] := -1, [11] := -1, [12] := -1, [13] := -1, [14] := -1, [15] := -1, [16] := -1, [17] := -1, [18] := -1, [19] := -1, [20] := -1, [21] := -1, [22] := -1, [23] := -1, [24] := -1, [25] := -1, [26] := -1, [27] := -1, [28] := -1, [29] := -1, [30] := -1, [31] := -1, [32] := -1, [33] := -1, [34] := -1, [35] := -1, [36] := -1, [37] := -1, [38] := -1, [39] := -1, [40] := -1, [41] := -1, [42] := -1, [43] := -1, [44] := -1, [45] := -1, [46] := -1, [47] := -1, [48] := -1, [49] := -1, [50] := -1, [51] := -1, [52] := -1, [53] := -1, [54] := -1, [55] := -1, [56] := -1, [57] := -1, [58] := -1, [59] := -1,
        [60] := -1, [61] := -1, [62] := -1, [63] := -1, [64] := -1, [65] := -1, [66] := -1, [67] := -1, [68] := -1, [69] := -1, [70] := -1, [71] := -1, [72] := -1, [73] := -1, [74] := -1, [75] := -1, [76] := -1, [77] := -1, [78] := -1, [79] := -1, [80] := -1, [81] := -1, [82] := -1, [83] := -1, [84] := -1, [85] := -1, [86] := -1, [87] := -1, [88] := -1, [89] := -1, [90] := -1, [91] := -1, [92] := -1, [93] := -1, [94] := -1, [95] := -1, [96] := -1, [97] := -1, [98] := -1, [99] := -1, [100] := -1, [101] := -1, [102] := -1, [103] := -1, [104] := -1, [105] := -1, [106] := -1, [107] := -1, [108] := -1, [109] := -1, [110] := -1, [111] := -1, [112] := -1, [113] := -1, [114] := -1, [115] := -1, [116] := -1, [117] := -1, [118] := -1, [119] := -1,
        [120] := -1, [121] := -1, [122] := -1, [123] := -1, [124] := -1, [125] := -1, [126] := -1, [127] := -1, [128] := -1, [129] := -1, [130] := -1, [131] := -1, [132] := -1, [133] := -1, [134] := -1, [135] := -1, [136] := -1, [137] := -1, [138] := -1, [139] := -1, [140] := -1, [141] := -1, [142] := -1, [143] := -1, [144] := -1, [145] := -1, [146] := -1, [147] := -1, [148] := -1, [149] := -1, [150] := -1, [151] := -1, [152] := -1, [153] := -1, [154] := -1, [155] := -1, [156] := -1, [157] := -1, [158] := -1, [159] := -1, [160] := -1, [161] := -1, [162] := -1, [163] := -1, [164] := -1, [165] := -1, [166] := -1, [167] := -1, [168] := -1, [169] := -1, [170] := -1, [171] := -1, [172] := -1, [173] := -1, [174] := -1, [175] := -1, [176] := -1, [177] := -1, [178] := -1, [179] := -1,
        [180] := -1, [181] := -1, [182] := -1, [183] := -1, [184] := -1, [185] := -1, [186] := -1, [187] := -1, [188] := -1, [189] := -1, [190] := -1, [191] := -1, [192] := -1, [193] := -1, [194] := -1, [195] := -1, [196] := -1, [197] := -1, [198] := -1, [199] := -1, [200] := -1, [201] := -1, [202] := -1, [203] := -1, [204] := -1, [205] := -1, [206] := -1, [207] := -1, [208] := -1, [209] := -1, [210] := -1, [211] := -1, [212] := -1, [213] := -1, [214] := -1, [215] := -1, [216] := -1, [217] := -1, [218] := -1, [219] := -1, [220] := -1, [221] := -1, [222] := -1, [223] := -1, [224] := -1, [225] := -1, [226] := -1, [227] := -1, [228] := -1, [229] := -1, [230] := -1, [231] := -1, [232] := -1, [233] := -1, [234] := -1, [235] := -1, [236] := -1, [237] := -1, [238] := -1, [239] := -1,
        [240] := -1, [241] := -1, [242] := -1, [243] := -1, [244] := -1, [245] := -1, [246] := -1, [247] := -1, [248] := -1, [249] := -1, [250] := -1, [251] := -1, [252] := -1, [253] := -1, [254] := -1, [255] := -1, [256] := -1, [257] := -1, [258] := -1, [259] := -1, [260] := -1, [261] := -1, [262] := -1, [263] := -1, [264] := -1, [265] := -1, [266] := -1, [267] := -1, [268] := -1, [269] := -1, [270] := -1, [271] := -1, [272] := -1, [273] := -1, [274] := -1, [275] := -1, [276] := -1, [277] := -1, [278] := -1, [279] := -1, [280] := -1, [281] := -1, [282] := -1, [283] := -1, [284] := -1, [285] := -1, [286] := -1, [287] := -1, [288] := -1, [289] := -1, [290] := -1, [291] := -1, [292] := -1, [293] := -1, [294] := -1, [295] := -1, [296] := -1, [297] := -1, [298] := -1, [299] := -1,
        [300] := -1, [301] := -1); {constant}
   Init_Stats : BOOL := 1;
   ITOP : INT := 66;
   old_index : DINT := 30;
   Proc_ST1AB : BOOL;
   Proc_ST1BA : BOOL := 1;
   Proc_ST2AB : BOOL := 1;
   Proc_ST2BA : BOOL;
   Qavg : REAL := 17.23263;
   Qmax : REAL := 19.713;
   Qmin : REAL := -17.572;
   QnC : REAL := 19.132;
   QpC : DINT := 19002;
   Qstd : REAL := 5045.6396;
   Qvar : REAL := 25.901094;
   Rbit : BOOL := 1;
   REbit : BOOL;
   SSID : STRING := 'D72F2CAC'; {access Read Only}
   SSID_Exists : INT := 1; {access Read Only}
   SSID_Locked : INT := 1; {access Read Only}
   ST1_HCntr : REAL := 0.58;
   ST1_QAB_INDX : INT[500] := ([0] := 30, [1] := 30, [2] := 30, [3] := 30, [4] := 30, [5] := 30, [6] := 30, [7] := 30, [8] := 30, [9] := 30, [10] := 30, [11] := 30, [12] := 30, [13] := 30, [14] := 30, [15] := 30, [16] := 30, [17] := 30, [18] := 30, [19] := 30, [20] := 30, [21] := 30, [22] := 30, [23] := 30, [24] := 30, [25] := 30, [26] := 30, [27] := 30, [28] := 30, [29] := 30, [30] := 30, [31] := 30, [32] := 30, [33] := 30, [34] := 30, [35] := 30, [36] := 30, [37] := 30, [38] := 30, [39] := 30, [40] := 30, [41] := 30, [42] := 30, [43] := 30, [44] := 30, [45] := 30, [46] := 30, [47] := 30, [48] := 30, [49] := 30, [50] := 30, [51] := 30, [52] := 30, [53] := 30, [54] := 30, [55] := 30, [56] := 30, [57] := 30, [58] := 30, [59] := 30,
        [60] := 30, [61] := 30, [62] := 30, [63] := 30, [64] := 30, [65] := 30, [66] := 30, [67] := 30, [68] := 30, [69] := 30, [70] := 30, [71] := 30, [72] := 30, [73] := 30, [74] := 30, [75] := 30, [76] := 30, [77] := 30, [78] := 30, [79] := 30, [80] := 30, [81] := 30, [82] := 30, [83] := 30, [84] := 30, [85] := 30, [86] := 30, [87] := 30, [88] := 30, [89] := 30, [90] := 30, [91] := 30, [92] := 30, [93] := 30, [94] := 30, [95] := 30, [96] := 30, [97] := 30, [98] := 30, [99] := 30, [100] := 30, [101] := 30, [102] := 30, [103] := 30, [104] := 30, [105] := 30, [106] := 30, [107] := 30, [108] := 30, [109] := 30, [110] := 30, [111] := 30, [112] := 30, [113] := 30, [114] := 30, [115] := 30, [116] := 30, [117] := 30, [118] := 30, [119] := 30,
        [120] := 30, [121] := 30, [122] := 30, [123] := 30, [124] := 30, [125] := 30, [126] := 30, [127] := 30, [128] := 30, [129] := 30, [130] := 30, [131] := 30, [132] := 30, [133] := 30, [134] := 30, [135] := 30, [136] := 30, [137] := 30, [138] := 30, [139] := 30, [140] := 30, [141] := 30, [142] := 30, [143] := 30, [144] := 30, [145] := 30, [146] := 30, [147] := 30, [148] := 30, [149] := 30, [150] := 30, [151] := 30, [152] := 30, [153] := 30, [154] := 30, [155] := 30, [156] := 30, [157] := 30, [158] := 30, [159] := 30, [160] := 30, [161] := 30, [162] := 30, [163] := 30, [164] := 30, [165] := 30, [166] := 30, [167] := 30, [168] := 30, [169] := 30, [170] := 30, [171] := 30, [172] := 30, [173] := 30, [174] := 30, [175] := 30, [176] := 30, [177] := 30, [178] := 30, [179] := 30,
        [180] := 30, [181] := 30, [182] := 30, [183] := 30, [184] := 30, [185] := 30, [186] := 30, [187] := 30, [188] := 30, [189] := 30, [190] := 30, [191] := 30, [192] := 30, [193] := 30, [194] := 30, [195] := 30, [196] := 30, [197] := 30, [198] := 30, [199] := 30, [200] := -1, [201] := -1, [202] := -1, [203] := -1, [204] := -1, [205] := -1, [206] := -1, [207] := -1, [208] := -1, [209] := -1, [210] := -1, [211] := -1, [212] := -1, [213] := -1, [214] := -1, [215] := -1, [216] := -1, [217] := -1, [218] := -1, [219] := -1, [220] := -1, [221] := -1, [222] := -1, [223] := -1, [224] := -1, [225] := -1, [226] := -1, [227] := -1, [228] := -1, [229] := -1, [230] := -1, [231] := -1, [232] := -1, [233] := -1, [234] := -1, [235] := -1, [236] := -1, [237] := -1, [238] := -1, [239] := -1,
        [240] := -1, [241] := -1, [242] := -1, [243] := -1, [244] := -1, [245] := -1, [246] := -1, [247] := -1, [248] := -1, [249] := -1, [250] := -1, [251] := -1, [252] := -1, [253] := -1, [254] := -1, [255] := -1, [256] := -1, [257] := -1, [258] := -1, [259] := -1, [260] := -1, [261] := -1, [262] := -1, [263] := -1, [264] := -1, [265] := -1, [266] := -1, [267] := -1, [268] := -1, [269] := -1, [270] := -1, [271] := -1, [272] := -1, [273] := -1, [274] := -1, [275] := -1, [276] := -1, [277] := -1, [278] := -1, [279] := -1, [280] := -1, [281] := -1, [282] := -1, [283] := -1, [284] := -1, [285] := -1, [286] := -1, [287] := -1, [288] := -1, [289] := -1, [290] := -1, [291] := -1, [292] := -1, [293] := -1, [294] := -1, [295] := -1, [296] := -1, [297] := -1, [298] := -1, [299] := -1,
        [300] := -1, [301] := -1);
   ST1_QAB_INDX_TOP : INT := 65;
   ST1_QBA_INDX : INT[500] := ([0] := 30, [1] := 30, [2] := 30, [3] := 30, [4] := 30, [5] := 30, [6] := 30, [7] := 30, [8] := 30, [9] := 30, [10] := 30, [11] := 30, [12] := 30, [13] := 30, [14] := 30, [15] := 30, [16] := 30, [17] := 30, [18] := 30, [19] := 30, [20] := 30, [21] := 30, [22] := 30, [23] := 30, [24] := 30, [25] := 30, [26] := 30, [27] := 30, [28] := 30, [29] := 30, [30] := 30, [31] := 30, [32] := 30, [33] := 30, [34] := 30, [35] := 30, [36] := 30, [37] := 30, [38] := 30, [39] := 30, [40] := 30, [41] := 30, [42] := 30, [43] := 30, [44] := 30, [45] := 30, [46] := 30, [47] := 30, [48] := 30, [49] := 30, [50] := 30, [51] := 30, [52] := 30, [53] := 30, [54] := 30, [55] := 30, [56] := 30, [57] := 30, [58] := 30, [59] := 30,
        [60] := 30, [61] := 30, [62] := 30, [63] := 30, [64] := 30, [65] := 30, [66] := 30, [67] := 30, [68] := 30, [69] := 30, [70] := 30, [71] := 30, [72] := 30, [73] := 30, [74] := 30, [75] := 30, [76] := 30, [77] := 30, [78] := 30, [79] := 30, [80] := 30, [81] := 30, [82] := 30, [83] := 30, [84] := 30, [85] := 30, [86] := 30, [87] := 30, [88] := 30, [89] := 30, [90] := 30, [91] := 30, [92] := 30, [93] := 30, [94] := 30, [95] := 30, [96] := 30, [97] := 30, [98] := 30, [99] := 30, [100] := 30, [101] := 30, [102] := 30, [103] := 30, [104] := 30, [105] := 30, [106] := 30, [107] := 30, [108] := 30, [109] := 30, [110] := 30, [111] := 30, [112] := 30, [113] := 30, [114] := 30, [115] := 30, [116] := 30, [117] := 30, [118] := 30, [119] := 30,
        [120] := 30, [121] := 30, [122] := 30, [123] := 30, [124] := 30, [125] := 30, [126] := 30, [127] := 30, [128] := 30, [129] := 30, [130] := 30, [131] := 30, [132] := 30, [133] := 30, [134] := 30, [135] := 30, [136] := 30, [137] := 30, [138] := 30, [139] := 30, [140] := 30, [141] := 30, [142] := 30, [143] := 30, [144] := 30, [145] := 30, [146] := 30, [147] := 30, [148] := 30, [149] := 30, [150] := 30, [151] := 30, [152] := 30, [153] := 30, [154] := 30, [155] := 30, [156] := 30, [157] := 30, [158] := 30, [159] := 30, [160] := 30, [161] := 30, [162] := 30, [163] := 30, [164] := 30, [165] := 30, [166] := 30, [167] := 30, [168] := 30, [169] := 30, [170] := 30, [171] := 30, [172] := 30, [173] := 30, [174] := 30, [175] := 30, [176] := 30, [177] := 30, [178] := 30, [179] := 30,
        [180] := 30, [181] := 30, [182] := 30, [183] := 30, [184] := 30, [185] := 30, [186] := 30, [187] := 30, [188] := 30, [189] := 30, [190] := 30, [191] := 30, [192] := 30, [193] := 30, [194] := 30, [195] := 30, [196] := 30, [197] := 30, [198] := 30, [199] := 30, [200] := -1, [201] := -1, [202] := -1, [203] := -1, [204] := -1, [205] := -1, [206] := -1, [207] := -1, [208] := -1, [209] := -1, [210] := -1, [211] := -1, [212] := -1, [213] := -1, [214] := -1, [215] := -1, [216] := -1, [217] := -1, [218] := -1, [219] := -1, [220] := -1, [221] := -1, [222] := -1, [223] := -1, [224] := -1, [225] := -1, [226] := -1, [227] := -1, [228] := -1, [229] := -1, [230] := -1, [231] := -1, [232] := -1, [233] := -1, [234] := -1, [235] := -1, [236] := -1, [237] := -1, [238] := -1, [239] := -1,
        [240] := -1, [241] := -1, [242] := -1, [243] := -1, [244] := -1, [245] := -1, [246] := -1, [247] := -1, [248] := -1, [249] := -1, [250] := -1, [251] := -1, [252] := -1, [253] := -1, [254] := -1, [255] := -1, [256] := -1, [257] := -1, [258] := -1, [259] := -1, [260] := -1, [261] := -1, [262] := -1, [263] := -1, [264] := -1, [265] := -1, [266] := -1, [267] := -1, [268] := -1, [269] := -1, [270] := -1, [271] := -1, [272] := -1, [273] := -1, [274] := -1, [275] := -1, [276] := -1, [277] := -1, [278] := -1, [279] := -1, [280] := -1, [281] := -1, [282] := -1, [283] := -1, [284] := -1, [285] := -1, [286] := -1, [287] := -1, [288] := -1, [289] := -1, [290] := -1, [291] := -1, [292] := -1, [293] := -1, [294] := -1, [295] := -1, [296] := -1, [297] := -1, [298] := -1, [299] := -1,
        [300] := -1, [301] := -1);
   ST1_QBA_INDX_TOP : INT := 66;
   ST2_HCntr : REAL := 15.98;
   ST2_QAB_INDX : INT[500] := ([0] := 30, [1] := 30, [2] := 30, [3] := 30, [4] := 30, [5] := 30, [6] := 30, [7] := 30, [8] := 30, [9] := 30, [10] := 30, [11] := 30, [12] := 30, [13] := 30, [14] := 30, [15] := 30, [16] := 30, [17] := 30, [18] := 30, [19] := 30, [20] := 30, [21] := 30, [22] := 30, [23] := 30, [24] := 30, [25] := 30, [26] := 30, [27] := 30, [28] := 30, [29] := 30, [30] := 30, [31] := 30, [32] := 30, [33] := 30, [34] := 30, [35] := 30, [36] := 30, [37] := 30, [38] := 30, [39] := 30, [40] := 30, [41] := 30, [42] := 30, [43] := 30, [44] := 30, [45] := 30, [46] := 30, [47] := 30, [48] := 30, [49] := 30, [50] := 30, [51] := 30, [52] := 30, [53] := 30, [54] := 30, [55] := 30, [56] := 30, [57] := 30, [58] := 30, [59] := 30,
        [60] := 30, [61] := 30, [62] := 30, [63] := 30, [64] := 30, [65] := 30, [66] := 30, [67] := 30, [68] := 30, [69] := 30, [70] := 30, [71] := 30, [72] := 30, [73] := 30, [74] := 30, [75] := 30, [76] := 30, [77] := 30, [78] := 30, [79] := 30, [80] := 30, [81] := 30, [82] := 30, [83] := 30, [84] := 30, [85] := 30, [86] := 30, [87] := 30, [88] := 30, [89] := 30, [90] := 30, [91] := 30, [92] := 30, [93] := 30, [94] := 30, [95] := 30, [96] := 30, [97] := 30, [98] := 30, [99] := 30, [100] := 30, [101] := 30, [102] := 30, [103] := 30, [104] := 30, [105] := 30, [106] := 30, [107] := 30, [108] := 30, [109] := 30, [110] := 30, [111] := 30, [112] := 30, [113] := 30, [114] := 30, [115] := 30, [116] := 30, [117] := 30, [118] := 30, [119] := 30,
        [120] := 30, [121] := 30, [122] := 30, [123] := 30, [124] := 30, [125] := 30, [126] := 30, [127] := 30, [128] := 30, [129] := 30, [130] := 30, [131] := 30, [132] := 30, [133] := 30, [134] := 30, [135] := 30, [136] := 30, [137] := 30, [138] := 30, [139] := 30, [140] := 30, [141] := 30, [142] := 30, [143] := 30, [144] := 30, [145] := 30, [146] := 30, [147] := 30, [148] := 30, [149] := 30, [150] := 30, [151] := 30, [152] := 30, [153] := 30, [154] := 30, [155] := 30, [156] := 30, [157] := 30, [158] := 30, [159] := 30, [160] := 30, [161] := 30, [162] := 30, [163] := 30, [164] := 30, [165] := 30, [166] := 30, [167] := 30, [168] := 30, [169] := 30, [170] := 30, [171] := 30, [172] := 30, [173] := 30, [174] := 30, [175] := 30, [176] := 30, [177] := 30, [178] := 30, [179] := 30,
        [180] := 30, [181] := 30, [182] := 30, [183] := 30, [184] := 30, [185] := 30, [186] := 30, [187] := 30, [188] := 30, [189] := 30, [190] := 30, [191] := 30, [192] := 30, [193] := 30, [194] := 30, [195] := 30, [196] := 30, [197] := 30, [198] := 30, [199] := 30, [200] := -1, [201] := -1, [202] := -1, [203] := -1, [204] := -1, [205] := -1, [206] := -1, [207] := -1, [208] := -1, [209] := -1, [210] := -1, [211] := -1, [212] := -1, [213] := -1, [214] := -1, [215] := -1, [216] := -1, [217] := -1, [218] := -1, [219] := -1, [220] := -1, [221] := -1, [222] := -1, [223] := -1, [224] := -1, [225] := -1, [226] := -1, [227] := -1, [228] := -1, [229] := -1, [230] := -1, [231] := -1, [232] := -1, [233] := -1, [234] := -1, [235] := -1, [236] := -1, [237] := -1, [238] := -1, [239] := -1,
        [240] := -1, [241] := -1, [242] := -1, [243] := -1, [244] := -1, [245] := -1, [246] := -1, [247] := -1, [248] := -1, [249] := -1, [250] := -1, [251] := -1, [252] := -1, [253] := -1, [254] := -1, [255] := -1, [256] := -1, [257] := -1, [258] := -1, [259] := -1, [260] := -1, [261] := -1, [262] := -1, [263] := -1, [264] := -1, [265] := -1, [266] := -1, [267] := -1, [268] := -1, [269] := -1, [270] := -1, [271] := -1, [272] := -1, [273] := -1, [274] := -1, [275] := -1, [276] := -1, [277] := -1, [278] := -1, [279] := -1, [280] := -1, [281] := -1, [282] := -1, [283] := -1, [284] := -1, [285] := -1, [286] := -1, [287] := -1, [288] := -1, [289] := -1, [290] := -1, [291] := -1, [292] := -1, [293] := -1, [294] := -1, [295] := -1, [296] := -1, [297] := -1, [298] := -1, [299] := -1,
        [300] := -1, [301] := -1);
   ST2_QAB_INDX_TOP : INT := 66;
   ST2_QBA_INDX : INT[500] := ([0] := 30, [1] := 30, [2] := 30, [3] := 30, [4] := 30, [5] := 30, [6] := 30, [7] := 30, [8] := 30, [9] := 30, [10] := 30, [11] := 30, [12] := 30, [13] := 30, [14] := 30, [15] := 30, [16] := 30, [17] := 30, [18] := 30, [19] := 30, [20] := 30, [21] := 30, [22] := 30, [23] := 30, [24] := 30, [25] := 30, [26] := 30, [27] := 30, [28] := 30, [29] := 30, [30] := 30, [31] := 30, [32] := 30, [33] := 30, [34] := 30, [35] := 30, [36] := 30, [37] := 30, [38] := 30, [39] := 30, [40] := 30, [41] := 30, [42] := 30, [43] := 30, [44] := 30, [45] := 30, [46] := 30, [47] := 30, [48] := 30, [49] := 30, [50] := 30, [51] := 30, [52] := 30, [53] := 30, [54] := 30, [55] := 30, [56] := 30, [57] := 30, [58] := 30, [59] := 30,
        [60] := 30, [61] := 30, [62] := 30, [63] := 30, [64] := 30, [65] := 30, [66] := 30, [67] := 30, [68] := 30, [69] := 30, [70] := 30, [71] := 30, [72] := 30, [73] := 30, [74] := 30, [75] := 30, [76] := 30, [77] := 30, [78] := 30, [79] := 30, [80] := 30, [81] := 30, [82] := 30, [83] := 30, [84] := 30, [85] := 30, [86] := 30, [87] := 30, [88] := 30, [89] := 30, [90] := 30, [91] := 30, [92] := 30, [93] := 30, [94] := 30, [95] := 30, [96] := 30, [97] := 30, [98] := 30, [99] := 30, [100] := 30, [101] := 30, [102] := 30, [103] := 30, [104] := 30, [105] := 30, [106] := 30, [107] := 30, [108] := 30, [109] := 30, [110] := 30, [111] := 30, [112] := 30, [113] := 30, [114] := 30, [115] := 30, [116] := 30, [117] := 30, [118] := 30, [119] := 30,
        [120] := 30, [121] := 30, [122] := 30, [123] := 30, [124] := 30, [125] := 30, [126] := 30, [127] := 30, [128] := 30, [129] := 30, [130] := 30, [131] := 30, [132] := 30, [133] := 30, [134] := 30, [135] := 30, [136] := 30, [137] := 30, [138] := 30, [139] := 30, [140] := 30, [141] := 30, [142] := 30, [143] := 30, [144] := 30, [145] := 30, [146] := 30, [147] := 30, [148] := 30, [149] := 30, [150] := 30, [151] := 30, [152] := 30, [153] := 30, [154] := 30, [155] := 30, [156] := 30, [157] := 30, [158] := 30, [159] := 30, [160] := 30, [161] := 30, [162] := 30, [163] := 30, [164] := 30, [165] := 30, [166] := 30, [167] := 30, [168] := 30, [169] := 30, [170] := 30, [171] := 30, [172] := 30, [173] := 30, [174] := 30, [175] := 30, [176] := 30, [177] := 30, [178] := 30, [179] := 30,
        [180] := 30, [181] := 30, [182] := 30, [183] := 30, [184] := 30, [185] := 30, [186] := 30, [187] := 30, [188] := 30, [189] := 30, [190] := 30, [191] := 30, [192] := 30, [193] := 30, [194] := 30, [195] := 30, [196] := 30, [197] := 30, [198] := 30, [199] := 30, [200] := -1, [201] := -1, [202] := -1, [203] := -1, [204] := -1, [205] := -1, [206] := -1, [207] := -1, [208] := -1, [209] := -1, [210] := -1, [211] := -1, [212] := -1, [213] := -1, [214] := -1, [215] := -1, [216] := -1, [217] := -1, [218] := -1, [219] := -1, [220] := -1, [221] := -1, [222] := -1, [223] := -1, [224] := -1, [225] := -1, [226] := -1, [227] := -1, [228] := -1, [229] := -1, [230] := -1, [231] := -1, [232] := -1, [233] := -1, [234] := -1, [235] := -1, [236] := -1, [237] := -1, [238] := -1, [239] := -1,
        [240] := -1, [241] := -1, [242] := -1, [243] := -1, [244] := -1, [245] := -1, [246] := -1, [247] := -1, [248] := -1, [249] := -1, [250] := -1, [251] := -1, [252] := -1, [253] := -1, [254] := -1, [255] := -1, [256] := -1, [257] := -1, [258] := -1, [259] := -1, [260] := -1, [261] := -1, [262] := -1, [263] := -1, [264] := -1, [265] := -1, [266] := -1, [267] := -1, [268] := -1, [269] := -1, [270] := -1, [271] := -1, [272] := -1, [273] := -1, [274] := -1, [275] := -1, [276] := -1, [277] := -1, [278] := -1, [279] := -1, [280] := -1, [281] := -1, [282] := -1, [283] := -1, [284] := -1, [285] := -1, [286] := -1, [287] := -1, [288] := -1, [289] := -1, [290] := -1, [291] := -1, [292] := -1, [293] := -1, [294] := -1, [295] := -1, [296] := -1, [297] := -1, [298] := -1, [299] := -1,
        [300] := -1, [301] := -1);
   ST2_QBA_INDX_TOP : INT := 17;
   Stat_Size : INT := 200;
   z1 : DINT := 199;
   z2 : REAL := 201.46675;
   z3 : REAL := 5.0456395;
END_VAR

ROUTINE AB_Stats   (* ladder *)
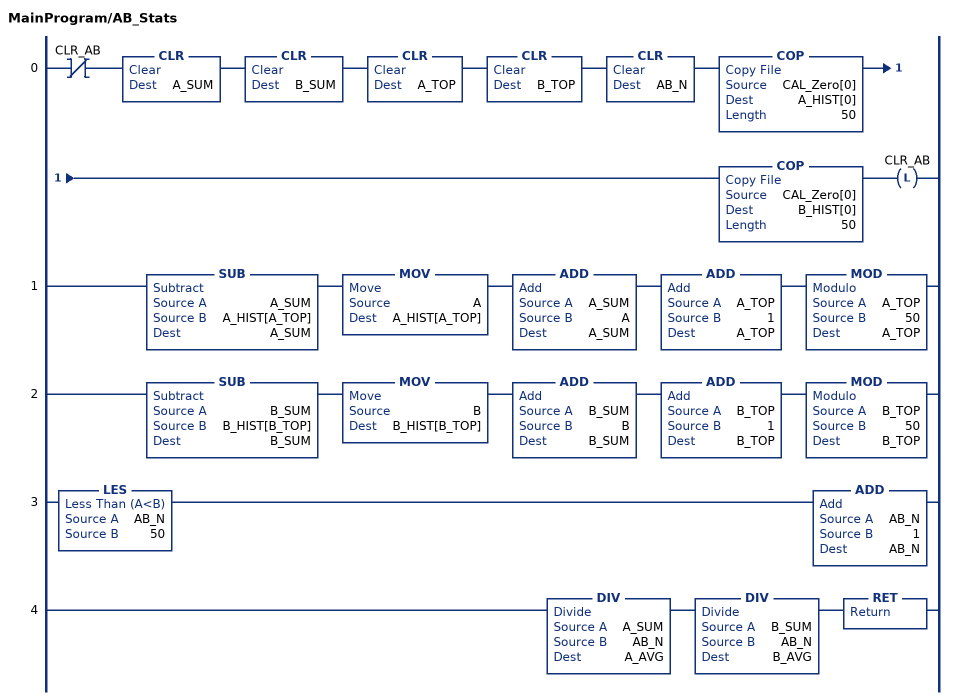
   0: XIO(CLR_AB)CLR(A_SUM)CLR(B_SUM)CLR(A_TOP)CLR(B_TOP)CLR(AB_N)COP(CAL_Zero[0],A_HIST[0],50)COP(CAL_Zero[0],B_HIST[0],50)OTL(CLR_AB);
   1: SUB(A_SUM,A_HIST[A_TOP],A_SUM)MOV(A,A_HIST[A_TOP])ADD(A_SUM,A,A_SUM)ADD(A_TOP,1,A_TOP)MOD(A_TOP,50,A_TOP);
   2: SUB(B_SUM,B_HIST[B_TOP],B_SUM)MOV(B,B_HIST[B_TOP])ADD(B_SUM,B,B_SUM)ADD(B_TOP,1,B_TOP)MOD(B_TOP,50,B_TOP);
   3: LES(AB_N,50)ADD(AB_N,1,AB_N);
   4: DIV(A_SUM,AB_N,A_AVG)DIV(B_SUM,AB_N,B_AVG)RET();
END_ROUTINE

ROUTINE Calc_Histogram   (* ladder *)
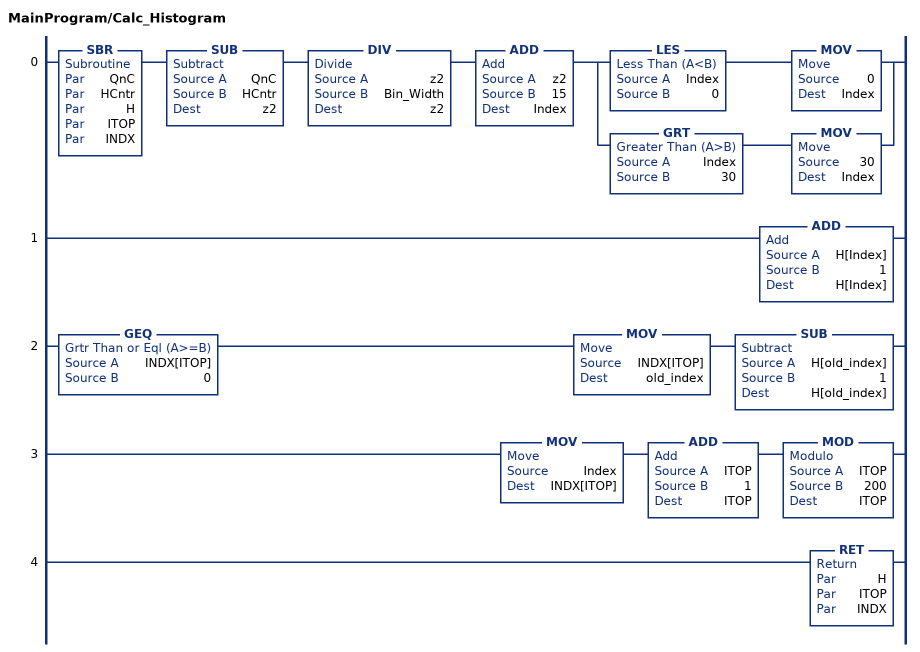
   0: SBR(QnC,HCntr,H,ITOP,INDX)SUB(QnC,HCntr,z2)DIV(z2,Bin_Width,z2)ADD(z2,15,Index)[LES(Index,0) MOV(0,Index) ,GRT(Index,30) MOV(30,Index) ];
   1: ADD(H[Index],1,H[Index]);
   2: GEQ(INDX[ITOP],0)MOV(INDX[ITOP],old_index)SUB(H[old_index],1,H[old_index]);
   3: MOV(Index,INDX[ITOP])ADD(ITOP,1,ITOP)MOD(ITOP,200,ITOP);
   4: RET(H,ITOP,INDX);
END_ROUTINE

ROUTINE Calc_Stats   (* ladder *)
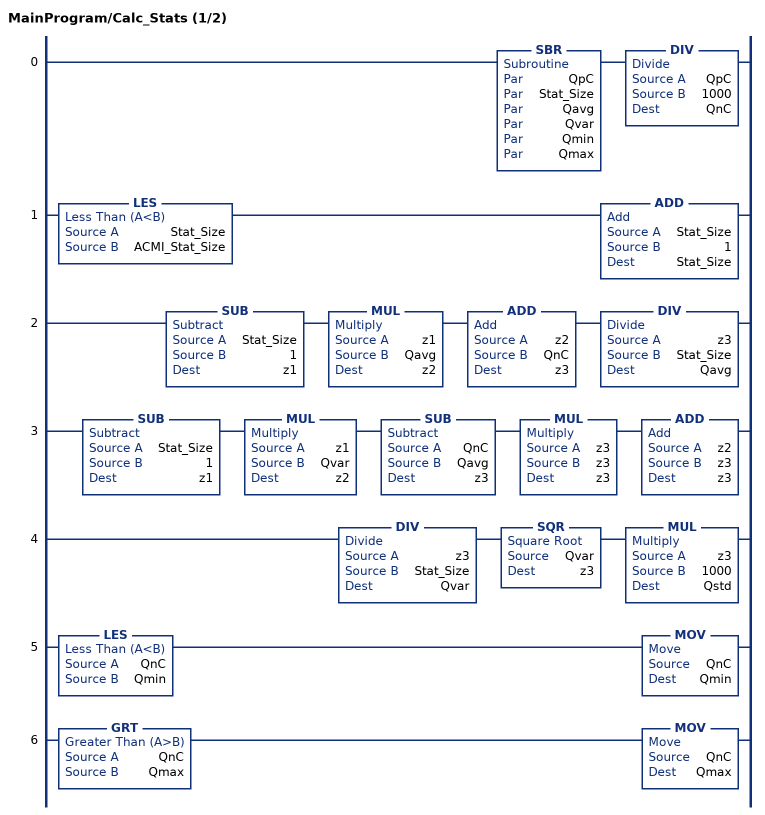
   0: SBR(QpC,Stat_Size,Qavg,Qvar,Qmin,Qmax)DIV(QpC,1000,QnC);
   1: LES(Stat_Size,ACMI_Stat_Size)ADD(Stat_Size,1,Stat_Size);
   2: SUB(Stat_Size,1,z1)MUL(z1,Qavg,z2)ADD(z2,QnC,z3)DIV(z3,Stat_Size,Qavg);
   3: SUB(Stat_Size,1,z1)MUL(z1,Qvar,z2)SUB(QnC,Qavg,z3)MUL(z3,z3,z3)ADD(z2,z3,z3);
   4: DIV(z3,Stat_Size,Qvar)SQR(Qvar,z3)MUL(z3,1000,Qstd);
   5: LES(QnC,Qmin)MOV(QnC,Qmin);
   6: GRT(QnC,Qmax)MOV(QnC,Qmax);
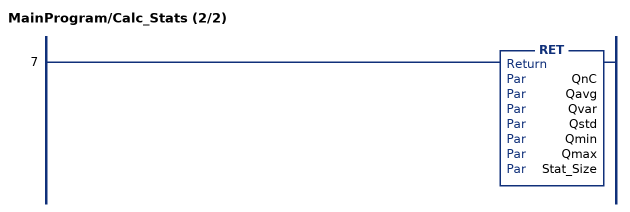
   7: RET(QnC,Qavg,Qvar,Qstd,Qmin,Qmax,Stat_Size);
END_ROUTINE
